// TIA Portal V16 export
// export: Created 2021-06-01T05:13:50.2237488Z, ExportSetting WithDefaults, DisplayName Totally Integrated Automation Portal, DisplayVersion V16 Update 4, DisplayName TIA Portal Version Control Interface, DisplayVersion V16 Update 2, DisplayName TIA Portal Openness, DisplayVersion V16 Update 4, DisplayName STEP 7 Professional, DisplayVersion V16 Update 4, DisplayName STEP 7 Safety, DisplayVersion V16, DisplayName WinCC Advanced, DisplayVersion V16 Update 4
FUNCTION "Demo" : Void   // FC2, F_FBD
{ S7_Optimized_Access := 'TRUE' }
VERSION : 0.1
// stored: AutoNumber true, IsIECCheckEnabled false, UDAEnableTagReadback false
   VAR_INPUT
      is_slow : Bool;
      left_clear : Bool;
      right_clear : Bool;
      mute_req : Bool;
      estop_clear : Bool;
   END_VAR
   VAR_OUTPUT
      stop : Bool;
   END_VAR
   VAR_TEMP
      mute_granted : Bool;
      scanners_ok : Bool;
   END_VAR
BEGIN

REGION Network 1
   // A mute request may be granted if the machine is moving slow enough to make it avoidable.
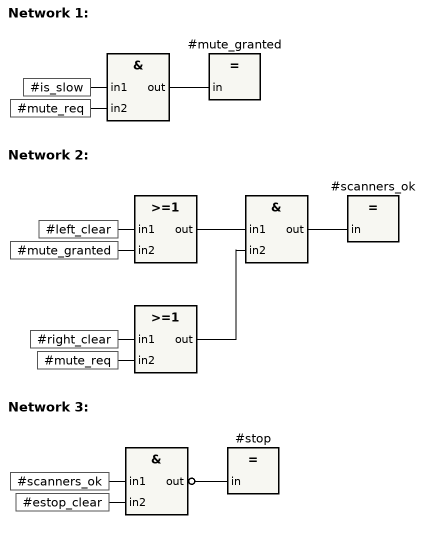
   #mute_granted := #is_slow AND #mute_req;
END_REGION

REGION Network 2
   // The safety scanner system evalutes the state of each safety field and condenses it to a single, overall status for the safety fields.
   #scanners_ok := (#left_clear OR #mute_granted) AND (#right_clear OR #mute_req);
END_REGION

REGION Network 3
   // Combine safety subsystems into a single stop variable
   #stop := NOT (#scanners_ok AND #estop_clear);
END_REGION
END_FUNCTION
